Xinje XDPPro project, PLC1: XDH-60T4 (software 3.7.17b 2023-10-13)

PROGRAM Ladder

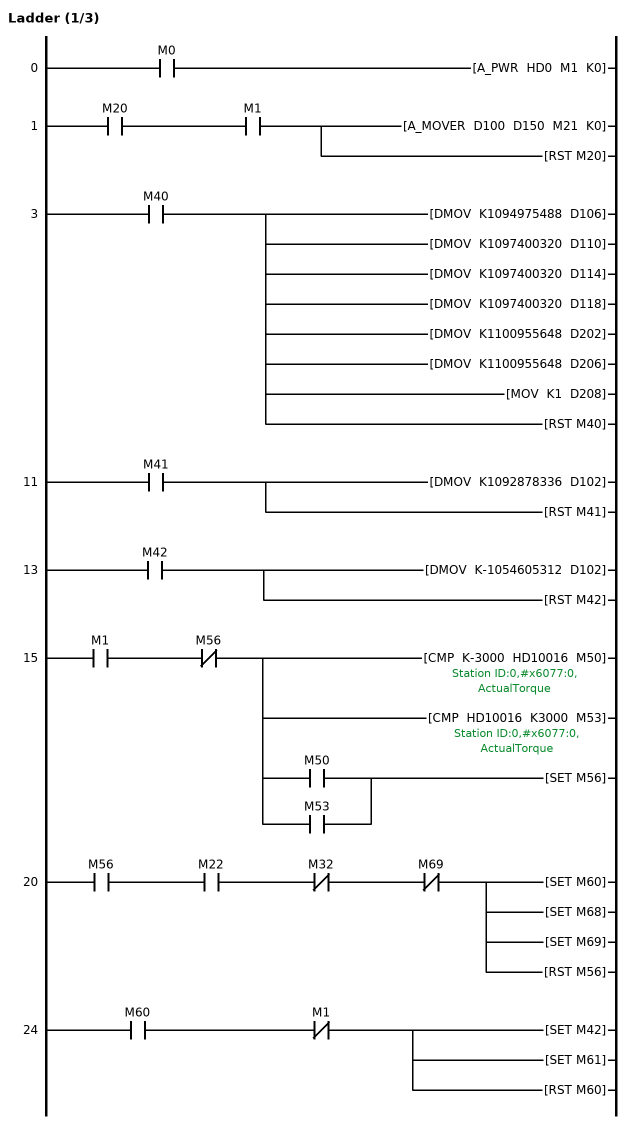
LD     M0
A_PWR  HD0 M1 K0
LD     M20
AND    M1
A_MOVER D100 D150 M21 K0
RST    M20
LD     M40
DMOV   K1094975488 D106
DMOV   K1097400320 D110
DMOV   K1097400320 D114
DMOV   K1097400320 D118
DMOV   K1100955648 D202
DMOV   K1100955648 D206
MOV    K1 D208
RST    M40
LD     M41
DMOV   K1092878336 D102
RST    M41
LD     M42
DMOV   K-1054605312 D102
RST    M42
LD     M1
ANI    M56
CMP    K-3000 HD10016 M50	; Station ID:0,#x6077:0,ActualTorque
CMP    HD10016 K3000 M53	; Station ID:0,#x6077:0,ActualTorque
LD     M50
OR     M53
ANB
SET    M56
LD     M56
AND    M22
ANI    M32
ANI    M69
SET    M60
SET    M68
SET    M69
RST    M56
LD     M60
ANI    M1
SET    M42
SET    M61
RST    M60

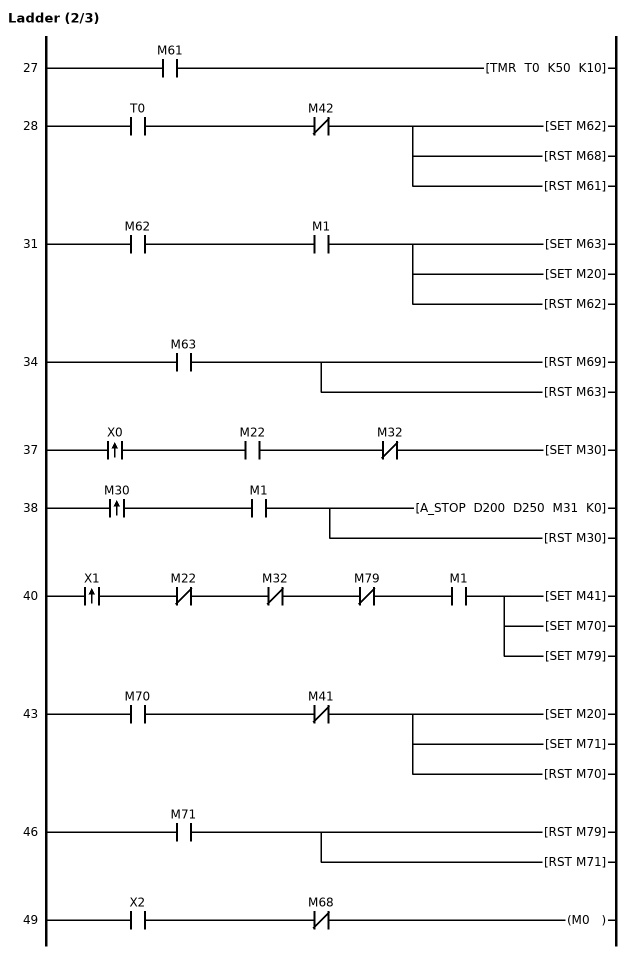
LD     M61
TMR    T0 K50 K10
LD     T0
ANI    M42
SET    M62
RST    M68
RST    M61
LD     M62
AND    M1
SET    M63
SET    M20
RST    M62
LD     M63
RST    M69
RST    M63
LDP    X0
AND    M22
ANI    M32
SET    M30
LDP    M30
AND    M1
A_STOP D200 D250 M31 K0
RST    M30
LDP    X1
ANI    M22
ANI    M32
ANI    M79
AND    M1
SET    M41
SET    M70
SET    M79
LD     M70
ANI    M41
SET    M20
SET    M71
RST    M70
LD     M71
RST    M79
RST    M71
LD     X2
ANI    M68
OUT    M0

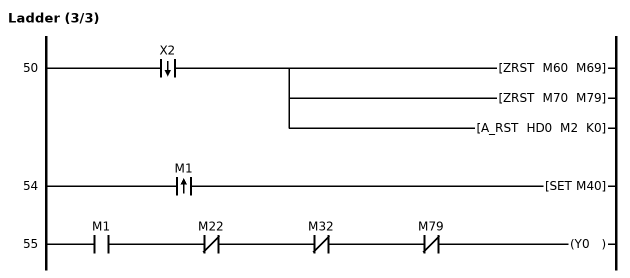
LDF    X2
ZRST   M60 M69
ZRST   M70 M79
A_RST  HD0 M2 K0
LDP    M1
SET    M40
LD     M1
ANI    M22
ANI    M32
ANI    M79
OUT    Y0

COMMENTS (devices not used above)
D20000	Axis 0:monitoring-The state machine
D20200	Axis 1:monitoring-The state machine
D20400	Axis 2:monitoring-The state machine
D20600	Axis 3:monitoring-The state machine
D20800	Axis 4:monitoring-The state machine
D21000	Axis 5:monitoring-The state machine
D21200	Axis 6:monitoring-The state machine
D21400	Axis 7:monitoring-The state machine
D21600	Axis 8:monitoring-The state machine
D21800	Axis 9:monitoring-The state machine
D22000	Axis 10:monitoring-The state machine
D22200	Axis 11:monitoring-The state machine
D22400	Axis 12:monitoring-The state machine
D22600	Axis 13:monitoring-The state machine
D22800	Axis 14:monitoring-The state machine
D23000	Axis 15:monitoring-The state machine
D23200	Axis 16:monitoring-The state machine
D23400	Axis 17:monitoring-The state machine
D23600	Axis 18:monitoring-The state machine
D23800	Axis 19:monitoring-The state machine
D24000	Axis 20:monitoring-The state machine
D24200	Axis 21:monitoring-The state machine
D24400	Axis 22:monitoring-The state machine
D24600	Axis 23:monitoring-The state machine
D24800	Axis 24:monitoring-The state machine
D25000	Axis 25:monitoring-The state machine
D25200	Axis 26:monitoring-The state machine
D25400	Axis 27:monitoring-The state machine
D25600	Axis 28:monitoring-The state machine
D25800	Axis 29:monitoring-The state machine
D26000	Axis 30:monitoring-The state machine
D26200	Axis 31:monitoring-The state machine
D20001	Axis 0:monitoring-Error code
D20201	Axis 1:monitoring-Error code
D20401	Axis 2:monitoring-Error code
D20601	Axis 3:monitoring-Error code
D20801	Axis 4:monitoring-Error code
D21001	Axis 5:monitoring-Error code
D21201	Axis 6:monitoring-Error code
D21401	Axis 7:monitoring-Error code
D21601	Axis 8:monitoring-Error code
D21801	Axis 9:monitoring-Error code
D22001	Axis 10:monitoring-Error code
D22201	Axis 11:monitoring-Error code
D22401	Axis 12:monitoring-Error code
D22601	Axis 13:monitoring-Error code
D22801	Axis 14:monitoring-Error code
D23001	Axis 15:monitoring-Error code
D23201	Axis 16:monitoring-Error code
D23401	Axis 17:monitoring-Error code
D23601	Axis 18:monitoring-Error code
D23801	Axis 19:monitoring-Error code
D24001	Axis 20:monitoring-Error code
D24201	Axis 21:monitoring-Error code
D24401	Axis 22:monitoring-Error code
D24601	Axis 23:monitoring-Error code
D24801	Axis 24:monitoring-Error code
D25001	Axis 25:monitoring-Error code
D25201	Axis 26:monitoring-Error code
D25401	Axis 27:monitoring-Error code
D25601	Axis 28:monitoring-Error code
D25801	Axis 29:monitoring-Error code
D26001	Axis 30:monitoring-Error code
D26201	Axis 31:monitoring-Error code
D20002	Axis 0:monitoring-Debug mode
D20202	Axis 1:monitoring-Debug mode
D20402	Axis 2:monitoring-Debug mode
D20602	Axis 3:monitoring-Debug mode
D20802	Axis 4:monitoring-Debug mode
D21002	Axis 5:monitoring-Debug mode
D21202	Axis 6:monitoring-Debug mode
D21402	Axis 7:monitoring-Debug mode
D21602	Axis 8:monitoring-Debug mode
D21802	Axis 9:monitoring-Debug mode
D22002	Axis 10:monitoring-Debug mode
D22202	Axis 11:monitoring-Debug mode
D22402	Axis 12:monitoring-Debug mode
D22602	Axis 13:monitoring-Debug mode
D22802	Axis 14:monitoring-Debug mode
D23002	Axis 15:monitoring-Debug mode
D23202	Axis 16:monitoring-Debug mode
D23402	Axis 17:monitoring-Debug mode
D23602	Axis 18:monitoring-Debug mode
D23802	Axis 19:monitoring-Debug mode
D24002	Axis 20:monitoring-Debug mode
D24202	Axis 21:monitoring-Debug mode
D24402	Axis 22:monitoring-Debug mode
D24602	Axis 23:monitoring-Debug mode
D24802	Axis 24:monitoring-Debug mode
D25002	Axis 25:monitoring-Debug mode
D25202	Axis 26:monitoring-Debug mode
D25402	Axis 27:monitoring-Debug mode
D25602	Axis 28:monitoring-Debug mode
D25802	Axis 29:monitoring-Debug mode
D26002	Axis 30:monitoring-Debug mode
D26202	Axis 31:monitoring-Debug mode
D20012	Axis 0:monitoring-The target location
D20212	Axis 1:monitoring-The target location
D20412	Axis 2:monitoring-The target location
D20612	Axis 3:monitoring-The target location
D20812	Axis 4:monitoring-The target location
D21012	Axis 5:monitoring-The target location
D21212	Axis 6:monitoring-The target location
D21412	Axis 7:monitoring-The target location
D21612	Axis 8:monitoring-The target location
D21812	Axis 9:monitoring-The target location
D22012	Axis 10:monitoring-The target location
D22212	Axis 11:monitoring-The target location
D22412	Axis 12:monitoring-The target location
D22612	Axis 13:monitoring-The target location
D22812	Axis 14:monitoring-The target location
D23012	Axis 15:monitoring-The target location
D23212	Axis 16:monitoring-The target location
D23412	Axis 17:monitoring-The target location
D23612	Axis 18:monitoring-The target location
D23812	Axis 19:monitoring-The target location
D24012	Axis 20:monitoring-The target location
D24212	Axis 21:monitoring-The target location
D24412	Axis 22:monitoring-The target location
D24612	Axis 23:monitoring-The target location
D24812	Axis 24:monitoring-The target location
D25012	Axis 25:monitoring-The target location
D25212	Axis 26:monitoring-The target location
D25412	Axis 27:monitoring-The target location
D25612	Axis 28:monitoring-The target location
D25812	Axis 29:monitoring-The target location
D26012	Axis 30:monitoring-The target location
D26212	Axis 31:monitoring-The target location
D20016	Axis 0:monitoring-Instruction position
D20216	Axis 1:monitoring-Instruction position
D20416	Axis 2:monitoring-Instruction position
D20616	Axis 3:monitoring-Instruction position
D20816	Axis 4:monitoring-Instruction position
D21016	Axis 5:monitoring-Instruction position
D21216	Axis 6:monitoring-Instruction position
D21416	Axis 7:monitoring-Instruction position
D21616	Axis 8:monitoring-Instruction position
D21816	Axis 9:monitoring-Instruction position
D22016	Axis 10:monitoring-Instruction position
D22216	Axis 11:monitoring-Instruction position
D22416	Axis 12:monitoring-Instruction position
D22616	Axis 13:monitoring-Instruction position
D22816	Axis 14:monitoring-Instruction position
D23016	Axis 15:monitoring-Instruction position
D23216	Axis 16:monitoring-Instruction position
D23416	Axis 17:monitoring-Instruction position
D23616	Axis 18:monitoring-Instruction position
D23816	Axis 19:monitoring-Instruction position
D24016	Axis 20:monitoring-Instruction position
D24216	Axis 21:monitoring-Instruction position
D24416	Axis 22:monitoring-Instruction position
D24616	Axis 23:monitoring-Instruction position
D24816	Axis 24:monitoring-Instruction position
D25016	Axis 25:monitoring-Instruction position
D25216	Axis 26:monitoring-Instruction position
D25416	Axis 27:monitoring-Instruction position
D25616	Axis 28:monitoring-Instruction position
D25816	Axis 29:monitoring-Instruction position
D26016	Axis 30:monitoring-Instruction position
D26216	Axis 31:monitoring-Instruction position
D20044	Axis 0:monitoring-Tatsächliche Position
D20244	Axis 1:monitoring-Tatsächliche Position
D20444	Axis 2:monitoring-Tatsächliche Position
D20644	Axis 3:monitoring-Tatsächliche Position
D20844	Axis 4:monitoring-Tatsächliche Position
D21044	Axis 5:monitoring-Tatsächliche Position
D21244	Axis 6:monitoring-Tatsächliche Position
D21444	Axis 7:monitoring-Tatsächliche Position
D21644	Axis 8:monitoring-Tatsächliche Position
D21844	Axis 9:monitoring-Tatsächliche Position
D22044	Axis 10:monitoring-Tatsächliche Position
D22244	Axis 11:monitoring-Tatsächliche Position
D22444	Axis 12:monitoring-Tatsächliche Position
D22644	Axis 13:monitoring-Tatsächliche Position
D22844	Axis 14:monitoring-Tatsächliche Position
D23044	Axis 15:monitoring-Tatsächliche Position
D23244	Axis 16:monitoring-Tatsächliche Position
D23444	Axis 17:monitoring-Tatsächliche Position
D23644	Axis 18:monitoring-Tatsächliche Position
D23844	Axis 19:monitoring-Tatsächliche Position
D24044	Axis 20:monitoring-Tatsächliche Position
D24244	Axis 21:monitoring-Tatsächliche Position
D24444	Axis 22:monitoring-Tatsächliche Position
D24644	Axis 23:monitoring-Tatsächliche Position
D24844	Axis 24:monitoring-Tatsächliche Position
D25044	Axis 25:monitoring-Tatsächliche Position
D25244	Axis 26:monitoring-Tatsächliche Position
D25444	Axis 27:monitoring-Tatsächliche Position
D25644	Axis 28:monitoring-Tatsächliche Position
D25844	Axis 29:monitoring-Tatsächliche Position
D26044	Axis 30:monitoring-Tatsächliche Position
D26244	Axis 31:monitoring-Tatsächliche Position
D20020	Axis 0:monitoring-Command speed
D20220	Axis 1:monitoring-Command speed
D20420	Axis 2:monitoring-Command speed
D20620	Axis 3:monitoring-Command speed
D20820	Axis 4:monitoring-Command speed
D21020	Axis 5:monitoring-Command speed
D21220	Axis 6:monitoring-Command speed
D21420	Axis 7:monitoring-Command speed
D21620	Axis 8:monitoring-Command speed
D21820	Axis 9:monitoring-Command speed
D22020	Axis 10:monitoring-Command speed
D22220	Axis 11:monitoring-Command speed
D22420	Axis 12:monitoring-Command speed
D22620	Axis 13:monitoring-Command speed
D22820	Axis 14:monitoring-Command speed
D23020	Axis 15:monitoring-Command speed
D23220	Axis 16:monitoring-Command speed
D23420	Axis 17:monitoring-Command speed
D23620	Axis 18:monitoring-Command speed
D23820	Axis 19:monitoring-Command speed
D24020	Axis 20:monitoring-Command speed
D24220	Axis 21:monitoring-Command speed
D24420	Axis 22:monitoring-Command speed
D24620	Axis 23:monitoring-Command speed
D24820	Axis 24:monitoring-Command speed
D25020	Axis 25:monitoring-Command speed
D25220	Axis 26:monitoring-Command speed
D25420	Axis 27:monitoring-Command speed
D25620	Axis 28:monitoring-Command speed
D25820	Axis 29:monitoring-Command speed
D26020	Axis 30:monitoring-Command speed
D26220	Axis 31:monitoring-Command speed
D20048	Axis 0:monitoring-Actual speed
D20248	Axis 1:monitoring-Actual speed
D20448	Axis 2:monitoring-Actual speed
D20648	Axis 3:monitoring-Actual speed
D20848	Axis 4:monitoring-Actual speed
D21048	Axis 5:monitoring-Actual speed
D21248	Axis 6:monitoring-Actual speed
D21448	Axis 7:monitoring-Actual speed
D21648	Axis 8:monitoring-Actual speed
D21848	Axis 9:monitoring-Actual speed
D22048	Axis 10:monitoring-Actual speed
D22248	Axis 11:monitoring-Actual speed
D22448	Axis 12:monitoring-Actual speed
D22648	Axis 13:monitoring-Actual speed
D22848	Axis 14:monitoring-Actual speed
D23048	Axis 15:monitoring-Actual speed
D23248	Axis 16:monitoring-Actual speed
D23448	Axis 17:monitoring-Actual speed
D23648	Axis 18:monitoring-Actual speed
D23848	Axis 19:monitoring-Actual speed
D24048	Axis 20:monitoring-Actual speed
D24248	Axis 21:monitoring-Actual speed
D24448	Axis 22:monitoring-Actual speed
D24648	Axis 23:monitoring-Actual speed
D24848	Axis 24:monitoring-Actual speed
D25048	Axis 25:monitoring-Actual speed
D25248	Axis 26:monitoring-Actual speed
D25448	Axis 27:monitoring-Actual speed
D25648	Axis 28:monitoring-Actual speed
D25848	Axis 29:monitoring-Actual speed
D26048	Axis 30:monitoring-Actual speed
D26248	Axis 31:monitoring-Actual speed
D20024	Axis 0:monitoring-Actual acceleration
D20224	Axis 1:monitoring-Actual acceleration
D20424	Axis 2:monitoring-Actual acceleration
D20624	Axis 3:monitoring-Actual acceleration
D20824	Axis 4:monitoring-Actual acceleration
D21024	Axis 5:monitoring-Actual acceleration
D21224	Axis 6:monitoring-Actual acceleration
D21424	Axis 7:monitoring-Actual acceleration
D21624	Axis 8:monitoring-Actual acceleration
D21824	Axis 9:monitoring-Actual acceleration
D22024	Axis 10:monitoring-Actual acceleration
D22224	Axis 11:monitoring-Actual acceleration
D22424	Axis 12:monitoring-Actual acceleration
D22624	Axis 13:monitoring-Actual acceleration
D22824	Axis 14:monitoring-Actual acceleration
D23024	Axis 15:monitoring-Actual acceleration
D23224	Axis 16:monitoring-Actual acceleration
D23424	Axis 17:monitoring-Actual acceleration
D23624	Axis 18:monitoring-Actual acceleration
D23824	Axis 19:monitoring-Actual acceleration
D24024	Axis 20:monitoring-Actual acceleration
D24224	Axis 21:monitoring-Actual acceleration
D24424	Axis 22:monitoring-Actual acceleration
D24624	Axis 23:monitoring-Actual acceleration
D24824	Axis 24:monitoring-Actual acceleration
D25024	Axis 25:monitoring-Actual acceleration
D25224	Axis 26:monitoring-Actual acceleration
D25424	Axis 27:monitoring-Actual acceleration
D25624	Axis 28:monitoring-Actual acceleration
D25824	Axis 29:monitoring-Actual acceleration
D26024	Axis 30:monitoring-Actual acceleration
D26224	Axis 31:monitoring-Actual acceleration
D20032	Axis 0:monitoring-Command torque
D20232	Axis 1:monitoring-Command torque
D20432	Axis 2:monitoring-Command torque
D20632	Axis 3:monitoring-Command torque
D20832	Axis 4:monitoring-Command torque
D21032	Axis 5:monitoring-Command torque
D21232	Axis 6:monitoring-Command torque
D21432	Axis 7:monitoring-Command torque
D21632	Axis 8:monitoring-Command torque
D21832	Axis 9:monitoring-Command torque
D22032	Axis 10:monitoring-Command torque
D22232	Axis 11:monitoring-Command torque
D22432	Axis 12:monitoring-Command torque
D22632	Axis 13:monitoring-Command torque
D22832	Axis 14:monitoring-Command torque
D23032	Axis 15:monitoring-Command torque
D23232	Axis 16:monitoring-Command torque
D23432	Axis 17:monitoring-Command torque
D23632	Axis 18:monitoring-Command torque
D23832	Axis 19:monitoring-Command torque
D24032	Axis 20:monitoring-Command torque
D24232	Axis 21:monitoring-Command torque
D24432	Axis 22:monitoring-Command torque
D24632	Axis 23:monitoring-Command torque
D24832	Axis 24:monitoring-Command torque
D25032	Axis 25:monitoring-Command torque
D25232	Axis 26:monitoring-Command torque
D25432	Axis 27:monitoring-Command torque
D25632	Axis 28:monitoring-Command torque
D25832	Axis 29:monitoring-Command torque
D26032	Axis 30:monitoring-Command torque
D26232	Axis 31:monitoring-Command torque
D20052	Axis 0:monitoring-Real-time torque
D20252	Axis 1:monitoring-Real-time torque
D20452	Axis 2:monitoring-Real-time torque
D20652	Axis 3:monitoring-Real-time torque
D20852	Axis 4:monitoring-Real-time torque
D21052	Axis 5:monitoring-Real-time torque
D21252	Axis 6:monitoring-Real-time torque
D21452	Axis 7:monitoring-Real-time torque
D21652	Axis 8:monitoring-Real-time torque
D21852	Axis 9:monitoring-Real-time torque
D22052	Axis 10:monitoring-Real-time torque
D22252	Axis 11:monitoring-Real-time torque
D22452	Axis 12:monitoring-Real-time torque
D22652	Axis 13:monitoring-Real-time torque
D22852	Axis 14:monitoring-Real-time torque
D23052	Axis 15:monitoring-Real-time torque
D23252	Axis 16:monitoring-Real-time torque
D23452	Axis 17:monitoring-Real-time torque
D23652	Axis 18:monitoring-Real-time torque
D23852	Axis 19:monitoring-Real-time torque
D24052	Axis 20:monitoring-Real-time torque
D24252	Axis 21:monitoring-Real-time torque
D24452	Axis 22:monitoring-Real-time torque
D24652	Axis 23:monitoring-Real-time torque
D24852	Axis 24:monitoring-Real-time torque
D25052	Axis 25:monitoring-Real-time torque
D25252	Axis 26:monitoring-Real-time torque
D25452	Axis 27:monitoring-Real-time torque
D25652	Axis 28:monitoring-Real-time torque
D25852	Axis 29:monitoring-Real-time torque
D26052	Axis 30:monitoring-Real-time torque
D26252	Axis 31:monitoring-Real-time torque
M20000	Axis 0:monitoring-Enabling state
M20050	Axis 1:monitoring-Enabling state
M20100	Axis 2:monitoring-Enabling state
M20150	Axis 3:monitoring-Enabling state
M20200	Axis 4:monitoring-Enabling state
M20250	Axis 5:monitoring-Enabling state
M20300	Axis 6:monitoring-Enabling state
M20350	Axis 7:monitoring-Enabling state
M20400	Axis 8:monitoring-Enabling state
M20450	Axis 9:monitoring-Enabling state
M20500	Axis 10:monitoring-Enabling state
M20550	Axis 11:monitoring-Enabling state
M20600	Axis 12:monitoring-Enabling state
M20650	Axis 13:monitoring-Enabling state
M20700	Axis 14:monitoring-Enabling state
M20750	Axis 15:monitoring-Enabling state
M20800	Axis 16:monitoring-Enabling state
M20850	Axis 17:monitoring-Enabling state
M20900	Axis 18:monitoring-Enabling state
M20950	Axis 19:monitoring-Enabling state
M21000	Axis 20:monitoring-Enabling state
M21050	Axis 21:monitoring-Enabling state
M21100	Axis 22:monitoring-Enabling state
M21150	Axis 23:monitoring-Enabling state
M21200	Axis 24:monitoring-Enabling state
M21250	Axis 25:monitoring-Enabling state
M21300	Axis 26:monitoring-Enabling state
M21350	Axis 27:monitoring-Enabling state
M21400	Axis 28:monitoring-Enabling state
M21450	Axis 29:monitoring-Enabling state
M21500	Axis 30:monitoring-Enabling state
M21550	Axis 31:monitoring-Enabling state
M20001	Axis 0:monitoring-Error status
M20051	Axis 1:monitoring-Error status
M20101	Axis 2:monitoring-Error status
M20151	Axis 3:monitoring-Error status
M20201	Axis 4:monitoring-Error status
M20251	Axis 5:monitoring-Error status
M20301	Axis 6:monitoring-Error status
M20351	Axis 7:monitoring-Error status
M20401	Axis 8:monitoring-Error status
M20451	Axis 9:monitoring-Error status
M20501	Axis 10:monitoring-Error status
M20551	Axis 11:monitoring-Error status
M20601	Axis 12:monitoring-Error status
M20651	Axis 13:monitoring-Error status
M20701	Axis 14:monitoring-Error status
M20751	Axis 15:monitoring-Error status
M20801	Axis 16:monitoring-Error status
M20851	Axis 17:monitoring-Error status
M20901	Axis 18:monitoring-Error status
M20951	Axis 19:monitoring-Error status
M21001	Axis 20:monitoring-Error status
M21051	Axis 21:monitoring-Error status
M21101	Axis 22:monitoring-Error status
M21151	Axis 23:monitoring-Error status
M21201	Axis 24:monitoring-Error status
M21251	Axis 25:monitoring-Error status
M21301	Axis 26:monitoring-Error status
M21351	Axis 27:monitoring-Error status
M21401	Axis 28:monitoring-Error status
M21451	Axis 29:monitoring-Error status
M21501	Axis 30:monitoring-Error status
M21551	Axis 31:monitoring-Error status
M20002	Axis 0:monitoring-Motion state
M20052	Axis 1:monitoring-Motion state
M20102	Axis 2:monitoring-Motion state
M20152	Axis 3:monitoring-Motion state
M20202	Axis 4:monitoring-Motion state
M20252	Axis 5:monitoring-Motion state
M20302	Axis 6:monitoring-Motion state
M20352	Axis 7:monitoring-Motion state
M20402	Axis 8:monitoring-Motion state
M20452	Axis 9:monitoring-Motion state
M20502	Axis 10:monitoring-Motion state
M20552	Axis 11:monitoring-Motion state
M20602	Axis 12:monitoring-Motion state
M20652	Axis 13:monitoring-Motion state
M20702	Axis 14:monitoring-Motion state
M20752	Axis 15:monitoring-Motion state
M20802	Axis 16:monitoring-Motion state
M20852	Axis 17:monitoring-Motion state
M20902	Axis 18:monitoring-Motion state
M20952	Axis 19:monitoring-Motion state
M21002	Axis 20:monitoring-Motion state
M21052	Axis 21:monitoring-Motion state
M21102	Axis 22:monitoring-Motion state
M21152	Axis 23:monitoring-Motion state
M21202	Axis 24:monitoring-Motion state
M21252	Axis 25:monitoring-Motion state
M21302	Axis 26:monitoring-Motion state
M21352	Axis 27:monitoring-Motion state
M21402	Axis 28:monitoring-Motion state
M21452	Axis 29:monitoring-Motion state
M21502	Axis 30:monitoring-Motion state
M21552	Axis 31:monitoring-Motion state
M20003	Axis 0:monitoring-Positioning state
M20053	Axis 1:monitoring-Positioning state
M20103	Axis 2:monitoring-Positioning state
M20153	Axis 3:monitoring-Positioning state
M20203	Axis 4:monitoring-Positioning state
M20253	Axis 5:monitoring-Positioning state
M20303	Axis 6:monitoring-Positioning state
M20353	Axis 7:monitoring-Positioning state
M20403	Axis 8:monitoring-Positioning state
M20453	Axis 9:monitoring-Positioning state
M20503	Axis 10:monitoring-Positioning state
M20553	Axis 11:monitoring-Positioning state
M20603	Axis 12:monitoring-Positioning state
M20653	Axis 13:monitoring-Positioning state
M20703	Axis 14:monitoring-Positioning state
M20753	Axis 15:monitoring-Positioning state
M20803	Axis 16:monitoring-Positioning state
M20853	Axis 17:monitoring-Positioning state
M20903	Axis 18:monitoring-Positioning state
M20953	Axis 19:monitoring-Positioning state
M21003	Axis 20:monitoring-Positioning state
M21053	Axis 21:monitoring-Positioning state
M21103	Axis 22:monitoring-Positioning state
M21153	Axis 23:monitoring-Positioning state
M21203	Axis 24:monitoring-Positioning state
M21253	Axis 25:monitoring-Positioning state
M21303	Axis 26:monitoring-Positioning state
M21353	Axis 27:monitoring-Positioning state
M21403	Axis 28:monitoring-Positioning state
M21453	Axis 29:monitoring-Positioning state
M21503	Axis 30:monitoring-Positioning state
M21553	Axis 31:monitoring-Positioning state
M20004	Axis 0:monitoring-home switch
M20054	Axis 1:monitoring-home switch
M20104	Axis 2:monitoring-home switch
M20154	Axis 3:monitoring-home switch
M20204	Axis 4:monitoring-home switch
M20254	Axis 5:monitoring-home switch
M20304	Axis 6:monitoring-home switch
M20354	Axis 7:monitoring-home switch
M20404	Axis 8:monitoring-home switch
M20454	Axis 9:monitoring-home switch
M20504	Axis 10:monitoring-home switch
M20554	Axis 11:monitoring-home switch
M20604	Axis 12:monitoring-home switch
M20654	Axis 13:monitoring-home switch
M20704	Axis 14:monitoring-home switch
M20754	Axis 15:monitoring-home switch
M20804	Axis 16:monitoring-home switch
M20854	Axis 17:monitoring-home switch
M20904	Axis 18:monitoring-home switch
M20954	Axis 19:monitoring-home switch
M21004	Axis 20:monitoring-home switch
M21054	Axis 21:monitoring-home switch
M21104	Axis 22:monitoring-home switch
M21154	Axis 23:monitoring-home switch
M21204	Axis 24:monitoring-home switch
M21254	Axis 25:monitoring-home switch
M21304	Axis 26:monitoring-home switch
M21354	Axis 27:monitoring-home switch
M21404	Axis 28:monitoring-home switch
M21454	Axis 29:monitoring-home switch
M21504	Axis 30:monitoring-home switch
M21554	Axis 31:monitoring-home switch
M20008	Axis 0:monitoring-Instruction completion status
M20058	Axis 1:monitoring-Instruction completion status
M20108	Axis 2:monitoring-Instruction completion status
M20158	Axis 3:monitoring-Instruction completion status
M20208	Axis 4:monitoring-Instruction completion status
M20258	Axis 5:monitoring-Instruction completion status
M20308	Axis 6:monitoring-Instruction completion status
M20358	Axis 7:monitoring-Instruction completion status
M20408	Axis 8:monitoring-Instruction completion status
M20458	Axis 9:monitoring-Instruction completion status
M20508	Axis 10:monitoring-Instruction completion status
M20558	Axis 11:monitoring-Instruction completion status
M20608	Axis 12:monitoring-Instruction completion status
M20658	Axis 13:monitoring-Instruction completion status
M20708	Axis 14:monitoring-Instruction completion status
M20758	Axis 15:monitoring-Instruction completion status
M20808	Axis 16:monitoring-Instruction completion status
M20858	Axis 17:monitoring-Instruction completion status
M20908	Axis 18:monitoring-Instruction completion status
M20958	Axis 19:monitoring-Instruction completion status
M21008	Axis 20:monitoring-Instruction completion status
M21058	Axis 21:monitoring-Instruction completion status
M21108	Axis 22:monitoring-Instruction completion status
M21158	Axis 23:monitoring-Instruction completion status
M21208	Axis 24:monitoring-Instruction completion status
M21258	Axis 25:monitoring-Instruction completion status
M21308	Axis 26:monitoring-Instruction completion status
M21358	Axis 27:monitoring-Instruction completion status
M21408	Axis 28:monitoring-Instruction completion status
M21458	Axis 29:monitoring-Instruction completion status
M21508	Axis 30:monitoring-Instruction completion status
M21558	Axis 31:monitoring-Instruction completion status
M20031	Axis 0:monitoring-positive software limit
M20081	Axis 1:monitoring-positive software limit
M20131	Axis 2:monitoring-positive software limit
M20181	Axis 3:monitoring-positive software limit
M20231	Axis 4:monitoring-positive software limit
M20281	Axis 5:monitoring-positive software limit
M20331	Axis 6:monitoring-positive software limit
M20381	Axis 7:monitoring-positive software limit
M20431	Axis 8:monitoring-positive software limit
M20481	Axis 9:monitoring-positive software limit
M20531	Axis 10:monitoring-positive software limit
M20581	Axis 11:monitoring-positive software limit
M20631	Axis 12:monitoring-positive software limit
M20681	Axis 13:monitoring-positive software limit
M20731	Axis 14:monitoring-positive software limit
M20781	Axis 15:monitoring-positive software limit
M20831	Axis 16:monitoring-positive software limit
M20881	Axis 17:monitoring-positive software limit
M20931	Axis 18:monitoring-positive software limit
M20981	Axis 19:monitoring-positive software limit
M21031	Axis 20:monitoring-positive software limit
M21081	Axis 21:monitoring-positive software limit
M21131	Axis 22:monitoring-positive software limit
M21181	Axis 23:monitoring-positive software limit
M21231	Axis 24:monitoring-positive software limit
M21281	Axis 25:monitoring-positive software limit
M21331	Axis 26:monitoring-positive software limit
M21381	Axis 27:monitoring-positive software limit
M21431	Axis 28:monitoring-positive software limit
M21481	Axis 29:monitoring-positive software limit
M21531	Axis 30:monitoring-positive software limit
M21581	Axis 31:monitoring-positive software limit
M20032	Axis 0:monitoring-negative software limit
M20082	Axis 1:monitoring-negative software limit
M20132	Axis 2:monitoring-negative software limit
M20182	Axis 3:monitoring-negative software limit
M20232	Axis 4:monitoring-negative software limit
M20282	Axis 5:monitoring-negative software limit
M20332	Axis 6:monitoring-negative software limit
M20382	Axis 7:monitoring-negative software limit
M20432	Axis 8:monitoring-negative software limit
M20482	Axis 9:monitoring-negative software limit
M20532	Axis 10:monitoring-negative software limit
M20582	Axis 11:monitoring-negative software limit
M20632	Axis 12:monitoring-negative software limit
M20682	Axis 13:monitoring-negative software limit
M20732	Axis 14:monitoring-negative software limit
M20782	Axis 15:monitoring-negative software limit
M20832	Axis 16:monitoring-negative software limit
M20882	Axis 17:monitoring-negative software limit
M20932	Axis 18:monitoring-negative software limit
M20982	Axis 19:monitoring-negative software limit
M21032	Axis 20:monitoring-negative software limit
M21082	Axis 21:monitoring-negative software limit
M21132	Axis 22:monitoring-negative software limit
M21182	Axis 23:monitoring-negative software limit
M21232	Axis 24:monitoring-negative software limit
M21282	Axis 25:monitoring-negative software limit
M21332	Axis 26:monitoring-negative software limit
M21382	Axis 27:monitoring-negative software limit
M21432	Axis 28:monitoring-negative software limit
M21482	Axis 29:monitoring-negative software limit
M21532	Axis 30:monitoring-negative software limit
M21582	Axis 31:monitoring-negative software limit
M20029	Axis 0:monitoring-positive hardware limit
M20079	Axis 1:monitoring-positive hardware limit
M20129	Axis 2:monitoring-positive hardware limit
M20179	Axis 3:monitoring-positive hardware limit
M20229	Axis 4:monitoring-positive hardware limit
M20279	Axis 5:monitoring-positive hardware limit
M20329	Axis 6:monitoring-positive hardware limit
M20379	Axis 7:monitoring-positive hardware limit
M20429	Axis 8:monitoring-positive hardware limit
M20479	Axis 9:monitoring-positive hardware limit
M20529	Axis 10:monitoring-positive hardware limit
M20579	Axis 11:monitoring-positive hardware limit
M20629	Axis 12:monitoring-positive hardware limit
M20679	Axis 13:monitoring-positive hardware limit
M20729	Axis 14:monitoring-positive hardware limit
M20779	Axis 15:monitoring-positive hardware limit
M20829	Axis 16:monitoring-positive hardware limit
M20879	Axis 17:monitoring-positive hardware limit
M20929	Axis 18:monitoring-positive hardware limit
M20979	Axis 19:monitoring-positive hardware limit
M21029	Axis 20:monitoring-positive hardware limit
M21079	Axis 21:monitoring-positive hardware limit
M21129	Axis 22:monitoring-positive hardware limit
M21179	Axis 23:monitoring-positive hardware limit
M21229	Axis 24:monitoring-positive hardware limit
M21279	Axis 25:monitoring-positive hardware limit
M21329	Axis 26:monitoring-positive hardware limit
M21379	Axis 27:monitoring-positive hardware limit
M21429	Axis 28:monitoring-positive hardware limit
M21479	Axis 29:monitoring-positive hardware limit
M21529	Axis 30:monitoring-positive hardware limit
M21579	Axis 31:monitoring-positive hardware limit
M20030	Axis 0:monitoring-negative hardware limit
M20080	Axis 1:monitoring-negative hardware limit
M20130	Axis 2:monitoring-negative hardware limit
M20180	Axis 3:monitoring-negative hardware limit
M20230	Axis 4:monitoring-negative hardware limit
M20280	Axis 5:monitoring-negative hardware limit
M20330	Axis 6:monitoring-negative hardware limit
M20380	Axis 7:monitoring-negative hardware limit
M20430	Axis 8:monitoring-negative hardware limit
M20480	Axis 9:monitoring-negative hardware limit
M20530	Axis 10:monitoring-negative hardware limit
M20580	Axis 11:monitoring-negative hardware limit
M20630	Axis 12:monitoring-negative hardware limit
M20680	Axis 13:monitoring-negative hardware limit
M20730	Axis 14:monitoring-negative hardware limit
M20780	Axis 15:monitoring-negative hardware limit
M20830	Axis 16:monitoring-negative hardware limit
M20880	Axis 17:monitoring-negative hardware limit
M20930	Axis 18:monitoring-negative hardware limit
M20980	Axis 19:monitoring-negative hardware limit
M21030	Axis 20:monitoring-negative hardware limit
M21080	Axis 21:monitoring-negative hardware limit
M21130	Axis 22:monitoring-negative hardware limit
M21180	Axis 23:monitoring-negative hardware limit
M21230	Axis 24:monitoring-negative hardware limit
M21280	Axis 25:monitoring-negative hardware limit
M21330	Axis 26:monitoring-negative hardware limit
M21380	Axis 27:monitoring-negative hardware limit
M21430	Axis 28:monitoring-negative hardware limit
M21480	Axis 29:monitoring-negative hardware limit
M21530	Axis 30:monitoring-negative hardware limit
M21580	Axis 31:monitoring-negative hardware limit
D20104	Axis 0:debugging-enable axis debug
D20304	Axis 1:debugging-enable axis debug
D20504	Axis 2:debugging-enable axis debug
D20704	Axis 3:debugging-enable axis debug
D20904	Axis 4:debugging-enable axis debug
D21104	Axis 5:debugging-enable axis debug
D21304	Axis 6:debugging-enable axis debug
D21504	Axis 7:debugging-enable axis debug
D21704	Axis 8:debugging-enable axis debug
D21904	Axis 9:debugging-enable axis debug
D22104	Axis 10:debugging-enable axis debug
D22304	Axis 11:debugging-enable axis debug
D22504	Axis 12:debugging-enable axis debug
D22704	Axis 13:debugging-enable axis debug
D22904	Axis 14:debugging-enable axis debug
D23104	Axis 15:debugging-enable axis debug
D23304	Axis 16:debugging-enable axis debug
D23504	Axis 17:debugging-enable axis debug
D23704	Axis 18:debugging-enable axis debug
D23904	Axis 19:debugging-enable axis debug
D24104	Axis 20:debugging-enable axis debug
D24304	Axis 21:debugging-enable axis debug
D24504	Axis 22:debugging-enable axis debug
D24704	Axis 23:debugging-enable axis debug
D24904	Axis 24:debugging-enable axis debug
D25104	Axis 25:debugging-enable axis debug
D25304	Axis 26:debugging-enable axis debug
D25504	Axis 27:debugging-enable axis debug
D25704	Axis 28:debugging-enable axis debug
D25904	Axis 29:debugging-enable axis debug
D26104	Axis 30:debugging-enable axis debug
D26304	Axis 31:debugging-enable axis debug
D20105	Axis 0:debugging-Movement type
D20305	Axis 1:debugging-Movement type
D20505	Axis 2:debugging-Movement type
D20705	Axis 3:debugging-Movement type
D20905	Axis 4:debugging-Movement type
D21105	Axis 5:debugging-Movement type
D21305	Axis 6:debugging-Movement type
D21505	Axis 7:debugging-Movement type
D21705	Axis 8:debugging-Movement type
D21905	Axis 9:debugging-Movement type
D22105	Axis 10:debugging-Movement type
D22305	Axis 11:debugging-Movement type
D22505	Axis 12:debugging-Movement type
D22705	Axis 13:debugging-Movement type
D22905	Axis 14:debugging-Movement type
D23105	Axis 15:debugging-Movement type
D23305	Axis 16:debugging-Movement type
D23505	Axis 17:debugging-Movement type
D23705	Axis 18:debugging-Movement type
D23905	Axis 19:debugging-Movement type
D24105	Axis 20:debugging-Movement type
D24305	Axis 21:debugging-Movement type
D24505	Axis 22:debugging-Movement type
D24705	Axis 23:debugging-Movement type
D24905	Axis 24:debugging-Movement type
D25105	Axis 25:debugging-Movement type
D25305	Axis 26:debugging-Movement type
D25505	Axis 27:debugging-Movement type
D25705	Axis 28:debugging-Movement type
D25905	Axis 29:debugging-Movement type
D26105	Axis 30:debugging-Movement type
D26305	Axis 31:debugging-Movement type
D20108	Axis 0:debugging-The target location
D20308	Axis 1:debugging-The target location
D20508	Axis 2:debugging-The target location
D20708	Axis 3:debugging-The target location
D20908	Axis 4:debugging-The target location
D21108	Axis 5:debugging-The target location
D21308	Axis 6:debugging-The target location
D21508	Axis 7:debugging-The target location
D21708	Axis 8:debugging-The target location
D21908	Axis 9:debugging-The target location
D22108	Axis 10:debugging-The target location
D22308	Axis 11:debugging-The target location
D22508	Axis 12:debugging-The target location
D22708	Axis 13:debugging-The target location
D22908	Axis 14:debugging-The target location
D23108	Axis 15:debugging-The target location
D23308	Axis 16:debugging-The target location
D23508	Axis 17:debugging-The target location
D23708	Axis 18:debugging-The target location
D23908	Axis 19:debugging-The target location
D24108	Axis 20:debugging-The target location
D24308	Axis 21:debugging-The target location
D24508	Axis 22:debugging-The target location
D24708	Axis 23:debugging-The target location
D24908	Axis 24:debugging-The target location
D25108	Axis 25:debugging-The target location
D25308	Axis 26:debugging-The target location
D25508	Axis 27:debugging-The target location
D25708	Axis 28:debugging-The target location
D25908	Axis 29:debugging-The target location
D26108	Axis 30:debugging-The target location
D26308	Axis 31:debugging-The target location
D20112	Axis 0:debugging-speed
D20312	Axis 1:debugging-speed
D20512	Axis 2:debugging-speed
D20712	Axis 3:debugging-speed
D20912	Axis 4:debugging-speed
D21112	Axis 5:debugging-speed
D21312	Axis 6:debugging-speed
D21512	Axis 7:debugging-speed
D21712	Axis 8:debugging-speed
D21912	Axis 9:debugging-speed
D22112	Axis 10:debugging-speed
D22312	Axis 11:debugging-speed
D22512	Axis 12:debugging-speed
D22712	Axis 13:debugging-speed
D22912	Axis 14:debugging-speed
D23112	Axis 15:debugging-speed
D23312	Axis 16:debugging-speed
D23512	Axis 17:debugging-speed
D23712	Axis 18:debugging-speed
D23912	Axis 19:debugging-speed
D24112	Axis 20:debugging-speed
D24312	Axis 21:debugging-speed
D24512	Axis 22:debugging-speed
D24712	Axis 23:debugging-speed
D24912	Axis 24:debugging-speed
D25112	Axis 25:debugging-speed
D25312	Axis 26:debugging-speed
D25512	Axis 27:debugging-speed
D25712	Axis 28:debugging-speed
D25912	Axis 29:debugging-speed
D26112	Axis 30:debugging-speed
D26312	Axis 31:debugging-speed
D20116	Axis 0:debugging-acceleration
D20316	Axis 1:debugging-acceleration
D20516	Axis 2:debugging-acceleration
D20716	Axis 3:debugging-acceleration
D20916	Axis 4:debugging-acceleration
D21116	Axis 5:debugging-acceleration
D21316	Axis 6:debugging-acceleration
D21516	Axis 7:debugging-acceleration
D21716	Axis 8:debugging-acceleration
D21916	Axis 9:debugging-acceleration
D22116	Axis 10:debugging-acceleration
D22316	Axis 11:debugging-acceleration
D22516	Axis 12:debugging-acceleration
D22716	Axis 13:debugging-acceleration
D22916	Axis 14:debugging-acceleration
D23116	Axis 15:debugging-acceleration
D23316	Axis 16:debugging-acceleration
D23516	Axis 17:debugging-acceleration
D23716	Axis 18:debugging-acceleration
D23916	Axis 19:debugging-acceleration
D24116	Axis 20:debugging-acceleration
D24316	Axis 21:debugging-acceleration
D24516	Axis 22:debugging-acceleration
D24716	Axis 23:debugging-acceleration
D24916	Axis 24:debugging-acceleration
D25116	Axis 25:debugging-acceleration
D25316	Axis 26:debugging-acceleration
D25516	Axis 27:debugging-acceleration
D25716	Axis 28:debugging-acceleration
D25916	Axis 29:debugging-acceleration
D26116	Axis 30:debugging-acceleration
D26316	Axis 31:debugging-acceleration
D20120	Axis 0:debugging-Reduce speed
D20320	Axis 1:debugging-Reduce speed
D20520	Axis 2:debugging-Reduce speed
D20720	Axis 3:debugging-Reduce speed
D20920	Axis 4:debugging-Reduce speed
D21120	Axis 5:debugging-Reduce speed
D21320	Axis 6:debugging-Reduce speed
D21520	Axis 7:debugging-Reduce speed
D21720	Axis 8:debugging-Reduce speed
D21920	Axis 9:debugging-Reduce speed
D22120	Axis 10:debugging-Reduce speed
D22320	Axis 11:debugging-Reduce speed
D22520	Axis 12:debugging-Reduce speed
D22720	Axis 13:debugging-Reduce speed
D22920	Axis 14:debugging-Reduce speed
D23120	Axis 15:debugging-Reduce speed
D23320	Axis 16:debugging-Reduce speed
D23520	Axis 17:debugging-Reduce speed
D23720	Axis 18:debugging-Reduce speed
D23920	Axis 19:debugging-Reduce speed
D24120	Axis 20:debugging-Reduce speed
D24320	Axis 21:debugging-Reduce speed
D24520	Axis 22:debugging-Reduce speed
D24720	Axis 23:debugging-Reduce speed
D24920	Axis 24:debugging-Reduce speed
D25120	Axis 25:debugging-Reduce speed
D25320	Axis 26:debugging-Reduce speed
D25520	Axis 27:debugging-Reduce speed
D25720	Axis 28:debugging-Reduce speed
D25920	Axis 29:debugging-Reduce speed
D26120	Axis 30:debugging-Reduce speed
D26320	Axis 31:debugging-Reduce speed
D20124	Axis 0:debugging-With the acceleration
D20324	Axis 1:debugging-With the acceleration
D20524	Axis 2:debugging-With the acceleration
D20724	Axis 3:debugging-With the acceleration
D20924	Axis 4:debugging-With the acceleration
D21124	Axis 5:debugging-With the acceleration
D21324	Axis 6:debugging-With the acceleration
D21524	Axis 7:debugging-With the acceleration
D21724	Axis 8:debugging-With the acceleration
D21924	Axis 9:debugging-With the acceleration
D22124	Axis 10:debugging-With the acceleration
D22324	Axis 11:debugging-With the acceleration
D22524	Axis 12:debugging-With the acceleration
D22724	Axis 13:debugging-With the acceleration
D22924	Axis 14:debugging-With the acceleration
D23124	Axis 15:debugging-With the acceleration
D23324	Axis 16:debugging-With the acceleration
D23524	Axis 17:debugging-With the acceleration
D23724	Axis 18:debugging-With the acceleration
D23924	Axis 19:debugging-With the acceleration
D24124	Axis 20:debugging-With the acceleration
D24324	Axis 21:debugging-With the acceleration
D24524	Axis 22:debugging-With the acceleration
D24724	Axis 23:debugging-With the acceleration
D24924	Axis 24:debugging-With the acceleration
D25124	Axis 25:debugging-With the acceleration
D25324	Axis 26:debugging-With the acceleration
D25524	Axis 27:debugging-With the acceleration
D25724	Axis 28:debugging-With the acceleration
D25924	Axis 29:debugging-With the acceleration
D26124	Axis 30:debugging-With the acceleration
D26324	Axis 31:debugging-With the acceleration
D20128	Axis 0:debugging-Modify position value
D20328	Axis 1:debugging-Modify position value
D20528	Axis 2:debugging-Modify position value
D20728	Axis 3:debugging-Modify position value
D20928	Axis 4:debugging-Modify position value
D21128	Axis 5:debugging-Modify position value
D21328	Axis 6:debugging-Modify position value
D21528	Axis 7:debugging-Modify position value
D21728	Axis 8:debugging-Modify position value
D21928	Axis 9:debugging-Modify position value
D22128	Axis 10:debugging-Modify position value
D22328	Axis 11:debugging-Modify position value
D22528	Axis 12:debugging-Modify position value
D22728	Axis 13:debugging-Modify position value
D22928	Axis 14:debugging-Modify position value
D23128	Axis 15:debugging-Modify position value
D23328	Axis 16:debugging-Modify position value
D23528	Axis 17:debugging-Modify position value
D23728	Axis 18:debugging-Modify position value
D23928	Axis 19:debugging-Modify position value
D24128	Axis 20:debugging-Modify position value
D24328	Axis 21:debugging-Modify position value
D24528	Axis 22:debugging-Modify position value
D24728	Axis 23:debugging-Modify position value
D24928	Axis 24:debugging-Modify position value
D25128	Axis 25:debugging-Modify position value
D25328	Axis 26:debugging-Modify position value
D25528	Axis 27:debugging-Modify position value
D25728	Axis 28:debugging-Modify position value
D25928	Axis 29:debugging-Modify position value
D26128	Axis 30:debugging-Modify position value
D26328	Axis 31:debugging-Modify position value
D20132	Axis 0:debugging-home offset
D20332	Axis 1:debugging-home offset
D20532	Axis 2:debugging-home offset
D20732	Axis 3:debugging-home offset
D20932	Axis 4:debugging-home offset
D21132	Axis 5:debugging-home offset
D21332	Axis 6:debugging-home offset
D21532	Axis 7:debugging-home offset
D21732	Axis 8:debugging-home offset
D21932	Axis 9:debugging-home offset
D22132	Axis 10:debugging-home offset
D22332	Axis 11:debugging-home offset
D22532	Axis 12:debugging-home offset
D22732	Axis 13:debugging-home offset
D22932	Axis 14:debugging-home offset
D23132	Axis 15:debugging-home offset
D23332	Axis 16:debugging-home offset
D23532	Axis 17:debugging-home offset
D23732	Axis 18:debugging-home offset
D23932	Axis 19:debugging-home offset
D24132	Axis 20:debugging-home offset
D24332	Axis 21:debugging-home offset
D24532	Axis 22:debugging-home offset
D24732	Axis 23:debugging-home offset
D24932	Axis 24:debugging-home offset
D25132	Axis 25:debugging-home offset
D25332	Axis 26:debugging-home offset
D25532	Axis 27:debugging-home offset
D25732	Axis 28:debugging-home offset
D25932	Axis 29:debugging-home offset
D26132	Axis 30:debugging-home offset
D26332	Axis 31:debugging-home offset
D20136	Axis 0:debugging-torque setting
D20336	Axis 1:debugging-torque setting
D20536	Axis 2:debugging-torque setting
D20736	Axis 3:debugging-torque setting
D20936	Axis 4:debugging-torque setting
D21136	Axis 5:debugging-torque setting
D21336	Axis 6:debugging-torque setting
D21536	Axis 7:debugging-torque setting
D21736	Axis 8:debugging-torque setting
D21936	Axis 9:debugging-torque setting
D22136	Axis 10:debugging-torque setting
D22336	Axis 11:debugging-torque setting
D22536	Axis 12:debugging-torque setting
D22736	Axis 13:debugging-torque setting
D22936	Axis 14:debugging-torque setting
D23136	Axis 15:debugging-torque setting
D23336	Axis 16:debugging-torque setting
D23536	Axis 17:debugging-torque setting
D23736	Axis 18:debugging-torque setting
D23936	Axis 19:debugging-torque setting
D24136	Axis 20:debugging-torque setting
D24336	Axis 21:debugging-torque setting
D24536	Axis 22:debugging-torque setting
D24736	Axis 23:debugging-torque setting
D24936	Axis 24:debugging-torque setting
D25136	Axis 25:debugging-torque setting
D25336	Axis 26:debugging-torque setting
D25536	Axis 27:debugging-torque setting
D25736	Axis 28:debugging-torque setting
D25936	Axis 29:debugging-torque setting
D26136	Axis 30:debugging-torque setting
D26336	Axis 31:debugging-torque setting
D20140	Axis 0:debugging-velocity limit
D20340	Axis 1:debugging-velocity limit
D20540	Axis 2:debugging-velocity limit
D20740	Axis 3:debugging-velocity limit
D20940	Axis 4:debugging-velocity limit
D21140	Axis 5:debugging-velocity limit
D21340	Axis 6:debugging-velocity limit
D21540	Axis 7:debugging-velocity limit
D21740	Axis 8:debugging-velocity limit
D21940	Axis 9:debugging-velocity limit
D22140	Axis 10:debugging-velocity limit
D22340	Axis 11:debugging-velocity limit
D22540	Axis 12:debugging-velocity limit
D22740	Axis 13:debugging-velocity limit
D22940	Axis 14:debugging-velocity limit
D23140	Axis 15:debugging-velocity limit
D23340	Axis 16:debugging-velocity limit
D23540	Axis 17:debugging-velocity limit
D23740	Axis 18:debugging-velocity limit
D23940	Axis 19:debugging-velocity limit
D24140	Axis 20:debugging-velocity limit
D24340	Axis 21:debugging-velocity limit
D24540	Axis 22:debugging-velocity limit
D24740	Axis 23:debugging-velocity limit
D24940	Axis 24:debugging-velocity limit
D25140	Axis 25:debugging-velocity limit
D25340	Axis 26:debugging-velocity limit
D25540	Axis 27:debugging-velocity limit
D25740	Axis 28:debugging-velocity limit
D25940	Axis 29:debugging-velocity limit
D26140	Axis 30:debugging-velocity limit
D26340	Axis 31:debugging-velocity limit
D20144	Axis 0:debugging-torque slope
D20344	Axis 1:debugging-torque slope
D20544	Axis 2:debugging-torque slope
D20744	Axis 3:debugging-torque slope
D20944	Axis 4:debugging-torque slope
D21144	Axis 5:debugging-torque slope
D21344	Axis 6:debugging-torque slope
D21544	Axis 7:debugging-torque slope
D21744	Axis 8:debugging-torque slope
D21944	Axis 9:debugging-torque slope
D22144	Axis 10:debugging-torque slope
D22344	Axis 11:debugging-torque slope
D22544	Axis 12:debugging-torque slope
D22744	Axis 13:debugging-torque slope
D22944	Axis 14:debugging-torque slope
D23144	Axis 15:debugging-torque slope
D23344	Axis 16:debugging-torque slope
D23544	Axis 17:debugging-torque slope
D23744	Axis 18:debugging-torque slope
D23944	Axis 19:debugging-torque slope
D24144	Axis 20:debugging-torque slope
D24344	Axis 21:debugging-torque slope
D24544	Axis 22:debugging-torque slope
D24744	Axis 23:debugging-torque slope
D24944	Axis 24:debugging-torque slope
D25144	Axis 25:debugging-torque slope
D25344	Axis 26:debugging-torque slope
D25544	Axis 27:debugging-torque slope
D25744	Axis 28:debugging-torque slope
D25944	Axis 29:debugging-torque slope
D26144	Axis 30:debugging-torque slope
D26344	Axis 31:debugging-torque slope
M20020	Axis 0:debugging-enable
M20070	Axis 1:debugging-enable
M20120	Axis 2:debugging-enable
M20170	Axis 3:debugging-enable
M20220	Axis 4:debugging-enable
M20270	Axis 5:debugging-enable
M20320	Axis 6:debugging-enable
M20370	Axis 7:debugging-enable
M20420	Axis 8:debugging-enable
M20470	Axis 9:debugging-enable
M20520	Axis 10:debugging-enable
M20570	Axis 11:debugging-enable
M20620	Axis 12:debugging-enable
M20670	Axis 13:debugging-enable
M20720	Axis 14:debugging-enable
M20770	Axis 15:debugging-enable
M20820	Axis 16:debugging-enable
M20870	Axis 17:debugging-enable
M20920	Axis 18:debugging-enable
M20970	Axis 19:debugging-enable
M21020	Axis 20:debugging-enable
M21070	Axis 21:debugging-enable
M21120	Axis 22:debugging-enable
M21170	Axis 23:debugging-enable
M21220	Axis 24:debugging-enable
M21270	Axis 25:debugging-enable
M21320	Axis 26:debugging-enable
M21370	Axis 27:debugging-enable
M21420	Axis 28:debugging-enable
M21470	Axis 29:debugging-enable
M21520	Axis 30:debugging-enable
M21570	Axis 31:debugging-enable
M20022	Axis 0:debugging-Target position motion
M20072	Axis 1:debugging-Target position motion
M20122	Axis 2:debugging-Target position motion
M20172	Axis 3:debugging-Target position motion
M20222	Axis 4:debugging-Target position motion
M20272	Axis 5:debugging-Target position motion
M20322	Axis 6:debugging-Target position motion
M20372	Axis 7:debugging-Target position motion
M20422	Axis 8:debugging-Target position motion
M20472	Axis 9:debugging-Target position motion
M20522	Axis 10:debugging-Target position motion
M20572	Axis 11:debugging-Target position motion
M20622	Axis 12:debugging-Target position motion
M20672	Axis 13:debugging-Target position motion
M20722	Axis 14:debugging-Target position motion
M20772	Axis 15:debugging-Target position motion
M20822	Axis 16:debugging-Target position motion
M20872	Axis 17:debugging-Target position motion
M20922	Axis 18:debugging-Target position motion
M20972	Axis 19:debugging-Target position motion
M21022	Axis 20:debugging-Target position motion
M21072	Axis 21:debugging-Target position motion
M21122	Axis 22:debugging-Target position motion
M21172	Axis 23:debugging-Target position motion
M21222	Axis 24:debugging-Target position motion
M21272	Axis 25:debugging-Target position motion
M21322	Axis 26:debugging-Target position motion
M21372	Axis 27:debugging-Target position motion
M21422	Axis 28:debugging-Target position motion
M21472	Axis 29:debugging-Target position motion
M21522	Axis 30:debugging-Target position motion
M21572	Axis 31:debugging-Target position motion
M20023	Axis 0:debugging-Positive point move
M20073	Axis 1:debugging-Positive point move
M20123	Axis 2:debugging-Positive point move
M20173	Axis 3:debugging-Positive point move
M20223	Axis 4:debugging-Positive point move
M20273	Axis 5:debugging-Positive point move
M20323	Axis 6:debugging-Positive point move
M20373	Axis 7:debugging-Positive point move
M20423	Axis 8:debugging-Positive point move
M20473	Axis 9:debugging-Positive point move
M20523	Axis 10:debugging-Positive point move
M20573	Axis 11:debugging-Positive point move
M20623	Axis 12:debugging-Positive point move
M20673	Axis 13:debugging-Positive point move
M20723	Axis 14:debugging-Positive point move
M20773	Axis 15:debugging-Positive point move
M20823	Axis 16:debugging-Positive point move
M20873	Axis 17:debugging-Positive point move
M20923	Axis 18:debugging-Positive point move
M20973	Axis 19:debugging-Positive point move
M21023	Axis 20:debugging-Positive point move
M21073	Axis 21:debugging-Positive point move
M21123	Axis 22:debugging-Positive point move
M21173	Axis 23:debugging-Positive point move
M21223	Axis 24:debugging-Positive point move
M21273	Axis 25:debugging-Positive point move
M21323	Axis 26:debugging-Positive point move
M21373	Axis 27:debugging-Positive point move
M21423	Axis 28:debugging-Positive point move
M21473	Axis 29:debugging-Positive point move
M21523	Axis 30:debugging-Positive point move
M21573	Axis 31:debugging-Positive point move
M20024	Axis 0:debugging-Reverse point move
M20074	Axis 1:debugging-Reverse point move
M20124	Axis 2:debugging-Reverse point move
M20174	Axis 3:debugging-Reverse point move
M20224	Axis 4:debugging-Reverse point move
M20274	Axis 5:debugging-Reverse point move
M20324	Axis 6:debugging-Reverse point move
M20374	Axis 7:debugging-Reverse point move
M20424	Axis 8:debugging-Reverse point move
M20474	Axis 9:debugging-Reverse point move
M20524	Axis 10:debugging-Reverse point move
M20574	Axis 11:debugging-Reverse point move
M20624	Axis 12:debugging-Reverse point move
M20674	Axis 13:debugging-Reverse point move
M20724	Axis 14:debugging-Reverse point move
M20774	Axis 15:debugging-Reverse point move
M20824	Axis 16:debugging-Reverse point move
M20874	Axis 17:debugging-Reverse point move
M20924	Axis 18:debugging-Reverse point move
M20974	Axis 19:debugging-Reverse point move
M21024	Axis 20:debugging-Reverse point move
M21074	Axis 21:debugging-Reverse point move
M21124	Axis 22:debugging-Reverse point move
M21174	Axis 23:debugging-Reverse point move
M21224	Axis 24:debugging-Reverse point move
M21274	Axis 25:debugging-Reverse point move
M21324	Axis 26:debugging-Reverse point move
M21374	Axis 27:debugging-Reverse point move
M21424	Axis 28:debugging-Reverse point move
M21474	Axis 29:debugging-Reverse point move
M21524	Axis 30:debugging-Reverse point move
M21574	Axis 31:debugging-Reverse point move
M20025	Axis 0:debugging-Back to the origin
M20075	Axis 1:debugging-Back to the origin
M20125	Axis 2:debugging-Back to the origin
M20175	Axis 3:debugging-Back to the origin
M20225	Axis 4:debugging-Back to the origin
M20275	Axis 5:debugging-Back to the origin
M20325	Axis 6:debugging-Back to the origin
M20375	Axis 7:debugging-Back to the origin
M20425	Axis 8:debugging-Back to the origin
M20475	Axis 9:debugging-Back to the origin
M20525	Axis 10:debugging-Back to the origin
M20575	Axis 11:debugging-Back to the origin
M20625	Axis 12:debugging-Back to the origin
M20675	Axis 13:debugging-Back to the origin
M20725	Axis 14:debugging-Back to the origin
M20775	Axis 15:debugging-Back to the origin
M20825	Axis 16:debugging-Back to the origin
M20875	Axis 17:debugging-Back to the origin
M20925	Axis 18:debugging-Back to the origin
M20975	Axis 19:debugging-Back to the origin
M21025	Axis 20:debugging-Back to the origin
M21075	Axis 21:debugging-Back to the origin
M21125	Axis 22:debugging-Back to the origin
M21175	Axis 23:debugging-Back to the origin
M21225	Axis 24:debugging-Back to the origin
M21275	Axis 25:debugging-Back to the origin
M21325	Axis 26:debugging-Back to the origin
M21375	Axis 27:debugging-Back to the origin
M21425	Axis 28:debugging-Back to the origin
M21475	Axis 29:debugging-Back to the origin
M21525	Axis 30:debugging-Back to the origin
M21575	Axis 31:debugging-Back to the origin
M20026	Axis 0:debugging-reset
M20076	Axis 1:debugging-reset
M20126	Axis 2:debugging-reset
M20176	Axis 3:debugging-reset
M20226	Axis 4:debugging-reset
M20276	Axis 5:debugging-reset
M20326	Axis 6:debugging-reset
M20376	Axis 7:debugging-reset
M20426	Axis 8:debugging-reset
M20476	Axis 9:debugging-reset
M20526	Axis 10:debugging-reset
M20576	Axis 11:debugging-reset
M20626	Axis 12:debugging-reset
M20676	Axis 13:debugging-reset
M20726	Axis 14:debugging-reset
M20776	Axis 15:debugging-reset
M20826	Axis 16:debugging-reset
M20876	Axis 17:debugging-reset
M20926	Axis 18:debugging-reset
M20976	Axis 19:debugging-reset
M21026	Axis 20:debugging-reset
M21076	Axis 21:debugging-reset
M21126	Axis 22:debugging-reset
M21176	Axis 23:debugging-reset
M21226	Axis 24:debugging-reset
M21276	Axis 25:debugging-reset
M21326	Axis 26:debugging-reset
M21376	Axis 27:debugging-reset
M21426	Axis 28:debugging-reset
M21476	Axis 29:debugging-reset
M21526	Axis 30:debugging-reset
M21576	Axis 31:debugging-reset
M20028	Axis 0:debugging-Modify the position
M20078	Axis 1:debugging-Modify the position
M20128	Axis 2:debugging-Modify the position
M20178	Axis 3:debugging-Modify the position
M20228	Axis 4:debugging-Modify the position
M20278	Axis 5:debugging-Modify the position
M20328	Axis 6:debugging-Modify the position
M20378	Axis 7:debugging-Modify the position
M20428	Axis 8:debugging-Modify the position
M20478	Axis 9:debugging-Modify the position
M20528	Axis 10:debugging-Modify the position
M20578	Axis 11:debugging-Modify the position
M20628	Axis 12:debugging-Modify the position
M20678	Axis 13:debugging-Modify the position
M20728	Axis 14:debugging-Modify the position
M20778	Axis 15:debugging-Modify the position
M20828	Axis 16:debugging-Modify the position
M20878	Axis 17:debugging-Modify the position
M20928	Axis 18:debugging-Modify the position
M20978	Axis 19:debugging-Modify the position
M21028	Axis 20:debugging-Modify the position
M21078	Axis 21:debugging-Modify the position
M21128	Axis 22:debugging-Modify the position
M21178	Axis 23:debugging-Modify the position
M21228	Axis 24:debugging-Modify the position
M21278	Axis 25:debugging-Modify the position
M21328	Axis 26:debugging-Modify the position
M21378	Axis 27:debugging-Modify the position
M21428	Axis 28:debugging-Modify the position
M21478	Axis 29:debugging-Modify the position
M21528	Axis 30:debugging-Modify the position
M21578	Axis 31:debugging-Modify the position